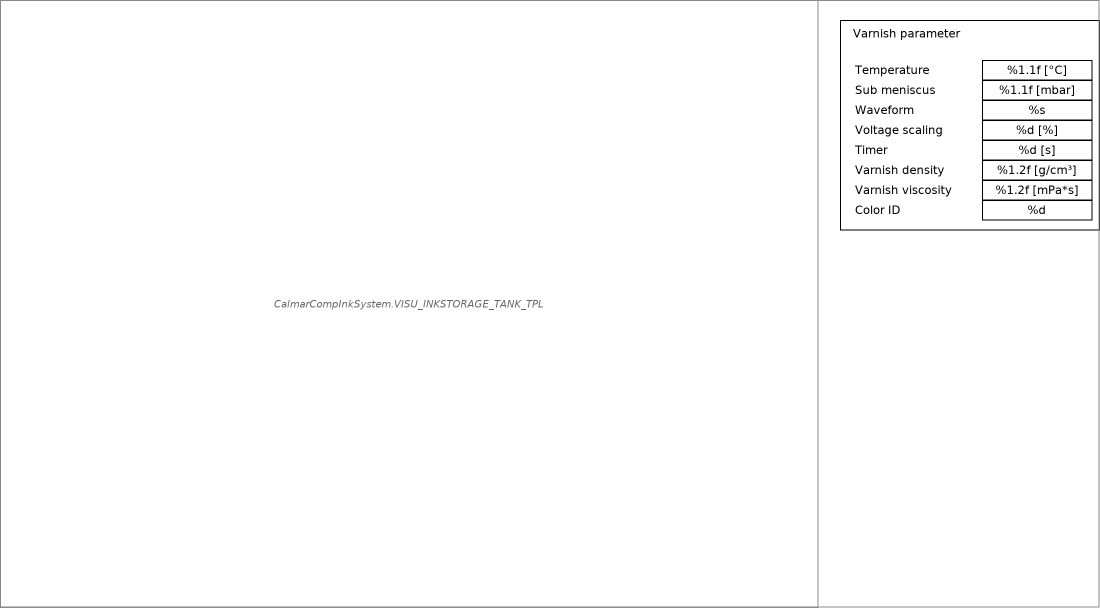
VISUALIZATION VISU_ADS_INKSTORAGE_TANK_DVT  // 1100x608
    Frame (0,0 818x608)
        shows CalmarCompInkSystem.VISU_INKSTORAGE_TANK_TPL(m_Idx_Max := CONFIGURATION.iCIk_NB_INKSTORAGE_TANK, m_ModId_StAdsStorageTank := PRG_INK.sAdsIkInkStorageTank[PRG_INK.iL_Sel_InkStorTank], m_Idx := PRG_INK.iL_Sel_InkStorTank, m_EnableBalanceLink := PRG_INK.bI_EnableBalanceLink, m_RefreshRate := PRG_INK.iI_RefreshRate, m_BalanceOffset := PRG_INK.fL_BalanceOffset[PRG_INK.iL_Sel_InkStorTank], m_CorrectionValue := PRG_INK.fI_CorrectionValue, m_MixerFeedbackExist := PRG_INK.bL_MixerFeedbackExist, m_MixerPulseIndicator := PRG_INK.bL_MixerPulseIndicator[PRG_INK.iL_Sel_InkStorTank], m_AckMixerPulseError := PRG_INK.bL_AckMixerPulseError[PRG_INK.iL_Sel_InkStorTank], m_MixerOnTime := PRG_INK.fL_MixerOnTime, m_MixerWaitTime := PRG_INK.fL_MixerWaitTime)
    Rectangle (840,20 260x210)
    Rectangle (982,60 110x20), "%1.1f [°C]", text variable: PRG_INK.sAdsIkInkStorageTank[PRG_INK.iL_Sel_InkStorTank].sI_InkParameter.sTemperature.fI_Val
        OnMouseDown: write the text variable via Edit, min PRG_INK.sAdsIkInkStorageTank[PRG_INK.iL_Sel_InkStorTank].sI_MaintenanceTimeout.lC_Min, max PRG_INK.sAdsIkInkStorageTank[PRG_INK.iL_Sel_InkStorTank].sI_MaintenanceTimeout.lC_Max
    Rectangle (852,60 130x20), "Temperature"
    Rectangle (850,25 191x17), "Varnish parameter"
    Rectangle (982,80 110x20), "%1.1f [mbar]", text variable: PRG_INK.sAdsIkInkStorageTank[PRG_INK.iL_Sel_InkStorTank].sI_InkParameter.sMeniscus.fI_Val
        OnMouseDown: write the text variable via Edit, min PRG_INK.sAdsIkInkStorageTank[PRG_INK.iL_Sel_InkStorTank].sI_InkParameter.sMeniscus.fC_Min, max PRG_INK.sAdsIkInkStorageTank[PRG_INK.iL_Sel_InkStorTank].sI_InkParameter.sMeniscus.fC_Max
    Rectangle (852,80 130x20), "Sub meniscus"
    Rectangle (982,100 110x20), "%s", text variable: PRG_INK.sAdsIkInkStorageTank[PRG_INK.iL_Sel_InkStorTank].sI_InkParameter.aWaveform
        OnMouseDown: write the text variable via Edit, min PRG_INK.sAdsIkInkStorageTank[PRG_INK.iL_Sel_InkStorTank].sI_MaintenanceTimeout.lC_Min, max PRG_INK.sAdsIkInkStorageTank[PRG_INK.iL_Sel_InkStorTank].sI_MaintenanceTimeout.lC_Max
    Rectangle (852,100 130x20), "Waveform"
    Rectangle (982,120 110x20), "%d [%]", text variable: PRG_INK.sAdsIkInkStorageTank[PRG_INK.iL_Sel_InkStorTank].sI_InkParameter.iVoltage
        OnMouseDown: write the text variable via Edit, min PRG_INK.sAdsIkInkStorageTank[PRG_INK.iL_Sel_InkStorTank].sI_MaintenanceTimeout.lC_Min, max PRG_INK.sAdsIkInkStorageTank[PRG_INK.iL_Sel_InkStorTank].sI_MaintenanceTimeout.lC_Max
    Rectangle (852,120 130x20), "Voltage scaling"
    Rectangle (982,140 110x20), "%d [s]", text variable: PRG_INK.sAdsIkInkStorageTank[PRG_INK.iL_Sel_InkStorTank].sI_InkParameter.iTimer
        OnMouseDown: write the text variable via Edit, min PRG_INK.sAdsIkInkStorageTank[PRG_INK.iL_Sel_InkStorTank].sI_MaintenanceTimeout.lC_Min, max PRG_INK.sAdsIkInkStorageTank[PRG_INK.iL_Sel_InkStorTank].sI_MaintenanceTimeout.lC_Max
    Rectangle (852,140 130x20), "Timer"
    Rectangle (982,160 110x20), "%1.2f [g/cm³]", text variable: PRG_INK.sAdsIkInkStorageTank[PRG_INK.iL_Sel_InkStorTank].sI_InkParameter.sDensity.fI_Val
        OnMouseDown: write the text variable via Edit, min PRG_INK.sAdsIkInkStorageTank[PRG_INK.iL_Sel_InkStorTank].sI_MaintenanceTimeout.lC_Min, max PRG_INK.sAdsIkInkStorageTank[PRG_INK.iL_Sel_InkStorTank].sI_MaintenanceTimeout.lC_Max
    Rectangle (852,160 130x20), "Varnish density"
    Rectangle (982,180 110x20), "%1.2f [mPa*s]", text variable: PRG_INK.sAdsIkInkStorageTank[PRG_INK.iL_Sel_InkStorTank].sI_InkParameter.sViscosity.fI_Val
        OnMouseDown: write the text variable via Edit, min PRG_INK.sAdsIkInkStorageTank[PRG_INK.iL_Sel_InkStorTank].sI_MaintenanceTimeout.lC_Min, max PRG_INK.sAdsIkInkStorageTank[PRG_INK.iL_Sel_InkStorTank].sI_MaintenanceTimeout.lC_Max
    Rectangle (852,180 130x20), "Varnish viscosity"
    Rectangle (982,200 110x20), "%d", text variable: PRG_INK.sAdsIkInkStorageTank[PRG_INK.iL_Sel_InkStorTank].sI_InkParameter.iColorId
        OnMouseDown: write the text variable via Edit, min PRG_INK.sAdsIkInkStorageTank[PRG_INK.iL_Sel_InkStorTank].sI_MaintenanceTimeout.lC_Min, max PRG_INK.sAdsIkInkStorageTank[PRG_INK.iL_Sel_InkStorTank].sI_MaintenanceTimeout.lC_Max
    Rectangle (852,200 130x20), "Color ID"
END_VISUALIZATION

(* stored: Version 1.1.0.1, ProductVersion 3.1.4024.11
   Visu VISU_ADS_INKSTORAGE_TANK_DVT: Id {28f0a6d8-dc87-4af0-90f2-96f8b1aab915} *)
